Omron CX-Programmer project NewProject (CX-Programmer 9.50)

# PLC NewPLC1: CP1E E20

## Global symbols (name address type ; comment)
0.00 BOOL  ; A/M
0.01 BOOL  ; PB Start
0.02 BOOL  ; detect part
0.03 BOOL  ; Metal Sensor
0.04 BOOL  ; non.met.post sensor
0.05 BOOL  ; met.post.sensor
0.06 BOOL  ; Pb Man M forw
0.07 BOOL  ; Pb Man M frev
0.08 BOOL  ; Pb Stop
100.00 BOOL  ; Auto Lamp
100.01 BOOL  ; Man Lp
100.02 BOOL  ; Met Lp
100.03 BOOL  ; Non Met Lp
100.04 BOOL  ; M.Forw
100.05 BOOL  ; M.Rev
W0.00 BOOL  ; Auto On
W0.01 BOOL  ; M.For ON
W0.02 BOOL  ; non.met.cond
W0.03 BOOL  ; met.cond
W0.04 BOOL  ; Stop M non metal
W0.05 BOOL  ; met.cond
W0.06 BOOL  ; stop M met
W0.07 BOOL  ; cut met.condition
W10.00 BOOL  ; srart auto
W10.01 BOOL  ; blink auto lamp
W20.00 BOOL  ; Stop Auto Process

## Program NewProgram1 (cyclic task 0)

### Section Section1

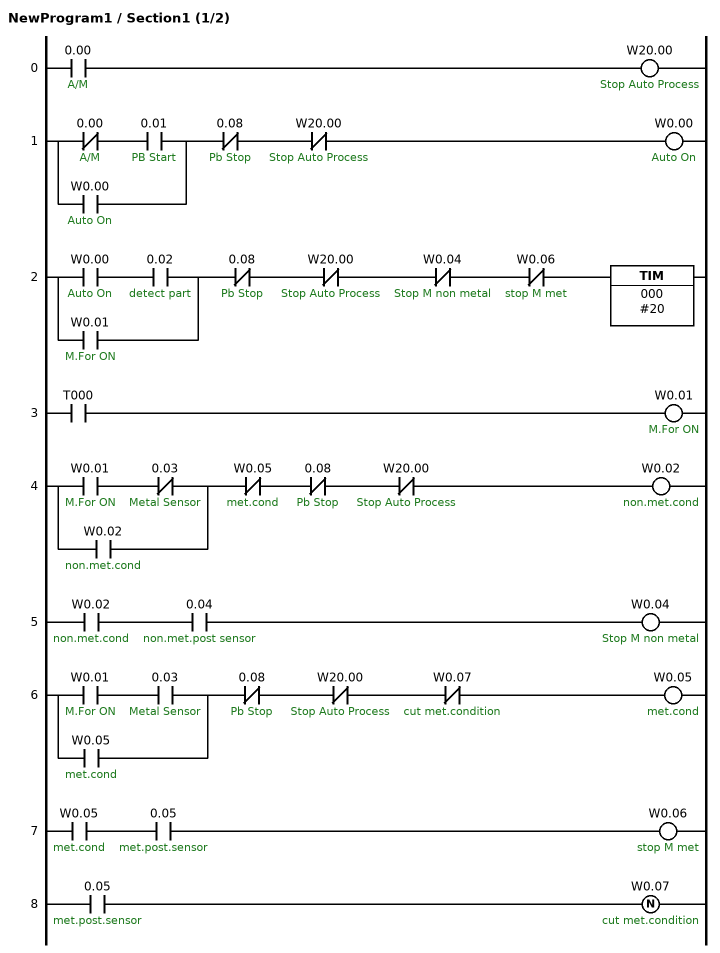
; rung 0
LD 0.00  ; A/M
OUT W20.00  ; Stop Auto Process
; rung 1
LDNOT 0.00  ; A/M
AND 0.01  ; PB Start
OR W0.00  ; Auto On
ANDNOT 0.08  ; Pb Stop
ANDNOT W20.00  ; Stop Auto Process
OUT W0.00  ; Auto On
; rung 2
LD W0.00  ; Auto On
AND 0.02  ; detect part
OR W0.01  ; M.For ON
ANDNOT 0.08  ; Pb Stop
ANDNOT W20.00  ; Stop Auto Process
ANDNOT W0.04  ; Stop M non metal
ANDNOT W0.06  ; stop M met
TIM 000 #20
; rung 3
LD T000
OUT W0.01  ; M.For ON
; rung 4
LD W0.01  ; M.For ON
ANDNOT 0.03  ; Metal Sensor
OR W0.02  ; non.met.cond
ANDNOT W0.05  ; met.cond
ANDNOT 0.08  ; Pb Stop
ANDNOT W20.00  ; Stop Auto Process
OUT W0.02  ; non.met.cond
; rung 5
LD W0.02  ; non.met.cond
AND 0.04  ; non.met.post sensor
OUT W0.04  ; Stop M non metal
; rung 6
LD W0.01  ; M.For ON
AND 0.03  ; Metal Sensor
OR W0.05  ; met.cond
ANDNOT 0.08  ; Pb Stop
ANDNOT W20.00  ; Stop Auto Process
ANDNOT W0.07  ; cut met.condition
OUT W0.05  ; met.cond
; rung 7
LD W0.05  ; met.cond
AND 0.05  ; met.post.sensor
OUT W0.06  ; stop M met
; rung 8
LD 0.05  ; met.post.sensor
DIFD(014) W0.07  ; cut met.condition

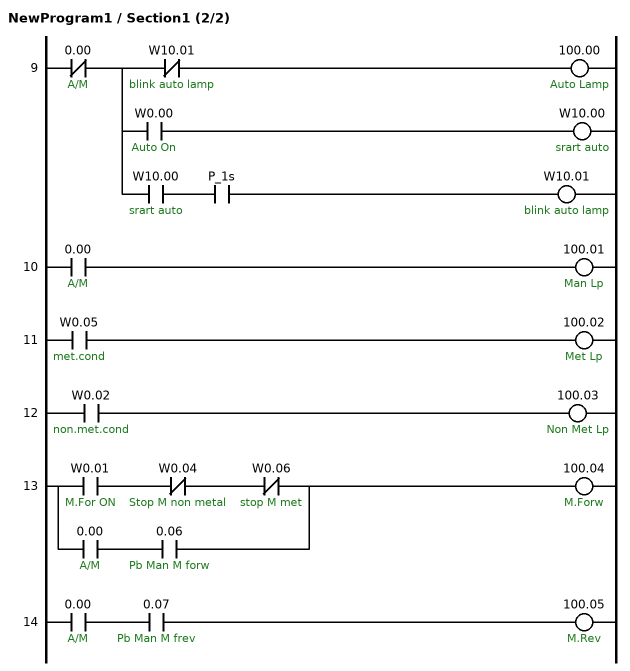
; rung 9
LDNOT 0.00  ; A/M
OUT TR0
ANDNOT W10.01  ; blink auto lamp
OUT 100.00  ; Auto Lamp
LD TR0
AND W0.00  ; Auto On
OUT W10.00  ; srart auto
LD TR0
AND W10.00  ; srart auto
AND P_1s
OUT W10.01  ; blink auto lamp
; rung 10
LD 0.00  ; A/M
OUT 100.01  ; Man Lp
; rung 11
LD W0.05  ; met.cond
OUT 100.02  ; Met Lp
; rung 12
LD W0.02  ; non.met.cond
OUT 100.03  ; Non Met Lp
; rung 13
LD W0.01  ; M.For ON
ANDNOT W0.04  ; Stop M non metal
ANDNOT W0.06  ; stop M met
LD 0.00  ; A/M
AND 0.06  ; Pb Man M forw
ORLD
OUT 100.04  ; M.Forw
; rung 14
LD 0.00  ; A/M
AND 0.07  ; Pb Man M frev
OUT 100.05  ; M.Rev

### Section END
; rung 0
END(001)